FUNCTION_BLOCK FB_CONTROL
VAR
	//Properties
	eControlMode		: CONTROL_MODE;
	stControlParameter	: CONTROL_PARAMETERS;
	
	fAct		:	REAL; 	// act value
	fSet		:	REAL; 	// set value
	fY			:	REAL; 	// control difference
	
	fbPID	:	FB_PID;
END_VAR

PROPERTY Act : REAL
GET
Act:=THIS^.fAct;
END_GET
SET
THIS^.fAct:=Act;
END_SET
END_PROPERTY

METHOD Control
VAR
	bResetController	: BOOL := FALSE;
END_VAR
IF fSet > 0 THEN
	bResetController := FALSE;
	// PID parameters are set in GVL 'ControlParameter_Props'
	fbPID(
		xSet := fSet,
		xAct := fAct,
		Kp := ControlParameter.Kp,
		Ti := ControlParameter.Ti,
		Td := ControlParameter.Td,
		LimLow := ControlParameter.LimLow,
		LimHigh := ControlParameter.LimHigh,
		bReverseActing := ControlParameter.bReverseActing,
		RST := bResetController,
		Y => fY
		);
ELSE
	IF NOT bResetController THEN
		bResetController := TRUE;
		fbPID(
		xSet := fSet,
		xAct := fAct,
		Kp := ControlParameter.Kp,
		Ti := ControlParameter.Ti,
		Td := ControlParameter.Td,
		LimLow := ControlParameter.LimLow,
		LimHigh := ControlParameter.LimHigh,
		bReverseActing := ControlParameter.bReverseActing,
		RST := bResetController,
		Y => fY
		);
	END_IF
	fY := 0;
END_IF
END_METHOD

PROPERTY ControlMode : CONTROL_MODE
GET
ControlMode := THIS^.eControlMode;
END_GET
SET
THIS^.eControlMode := ControlMode;
END_SET
END_PROPERTY

PROPERTY ControlParameter : REFERENCE TO CONTROL_PARAMETERS
GET
ControlParameter REF=THIS^.stControlParameter;
END_GET
SET
THIS^.stControlParameter := ControlParameter;
END_SET
END_PROPERTY

PROPERTY Set : REAL
GET
Set:=THIS^.fSet;
END_GET
SET
THIS^.fSet:=Set;
END_SET
END_PROPERTY

PROPERTY Y : Real
GET
Y :=THIS^.fY;
END_GET
END_PROPERTY

END_FUNCTION_BLOCK

(* stored: Version 1.1.0.1
   POU FB_CONTROL: Id {431e90c2-3f53-42b6-bdae-8ec16d6fc076}, SpecialFunc None
   Property Act: Id {a6fed756-94cb-4bc0-a5a3-e34d1122c3dc}
   Get Get: Id {bc5bfd96-0d2e-4c61-af4b-7ad245b56d05}
   Set Set: Id {ffe151c8-1d99-4325-909a-6869261acdec}
   Method Control: Id {083bf493-ca97-46cd-9a57-3b1f413e339b}
   Property ControlMode: Id {2c47d686-cebe-4be6-a87d-2ab633d6c170}
   Get Get: Id {9e8c2fc4-905b-4af9-8c5f-99472f167384}
   Set Set: Id {00cbe839-eed2-405b-9e38-2a0901f15eff}
   Property ControlParameter: Id {c0af4740-e9c7-4c8d-a4b6-02f0c80d2263}
   Get Get: Id {568e2ace-b184-49d3-8a23-9cdb68df5b59}
   Set Set: Id {bd990303-8953-45ff-ae9d-d763ab04462d}
   Property Set: Id {c4e9ea93-8bd6-4108-a270-e0516649d553}
   Get Get: Id {2bd4f9d1-926d-4013-ac44-46cefe45ff2a}
   Set Set: Id {b642650c-7e91-4fd2-acf5-56425ce13e9c}
   Property Y: Id {1f067d2a-11fc-4b84-96c4-bfc38f4f42d0}
   Get Get: Id {505434c3-90be-4e5c-8656-432b8d7caaac} *)
